FUNCTION_BLOCK LedLamp
VAR
	output AT %Q* : BOOL;
END_VAR

METHOD Off
VAR_INPUT
END_VAR
output := FALSE;
END_METHOD

METHOD On
VAR_INPUT
END_VAR
output := TRUE;
END_METHOD

END_FUNCTION_BLOCK

(* stored: Version 1.1.0.1, ProductVersion 3.1.4024.12
   POU LedLamp: Id {2e882cf5-3d00-4221-9a19-847a0714e3aa}, SpecialFunc None
   Method Off: Id {da7ba108-a618-4aa5-a0cf-d6e8d2016649}
   Method On: Id {e562fba0-efa2-4bb1-b9fe-3b9ec4fb4e2e} *)
